FUNCTION FUN_HOMING : BOOL
VAR_INPUT
END_VAR
VAR
END_VAR

END_FUNCTION

(* stored: Version 1.1.0.1, ProductVersion 3.1.4024.12
   POU FUN_HOMING: Id {c8dc9b93-a2c3-4e83-ba78-da6aa376e3ce}, SpecialFunc None *)
